// TwinCAT 3 PLC project Lectures
// ProgramVersion: 3.1.4024.0
// libraries:
//   Tc2_Standard, * (Beckhoff Automation GmbH)
//   Tc2_System, * (Beckhoff Automation GmbH)
//   Tc3_Module, * (Beckhoff Automation GmbH)
// project tree:
//   DUTs/ Motor.TcTLEO (not stored), Movement.TcTLEO, MovementDirection.TcTLEO (not stored), Recipe.TcDUT
//   GVLs/ Automatic.TcGVL, IO.TcGVL (not stored)
//   / PlcTask.TcTTO (not stored)
//   POUs/ AutomaticControl.TcPOU (not stored), CountCurrentPosition.TcPOU, ExecuteCurrentRecipe.TcPOU (not stored), Initialize.TcPOU, MakeNewRecipe.TcPOU (not stored), ManualControl.TcPOU, MAIN.TcPOU, MotorSelection.TcPOU (not stored), Recipe1.TcPOU (not stored), Recipe2.TcPOU, RestorePreviousAutomaticState.TcPOU, Safety.TcPOU (not stored)
//   POUs/Lectures%27 programs/ p00_true_false.TcPOU (not stored), p01_sequential.TcPOU (not stored), p02_clock.TcPOU (not stored), p03_SR1.TcPOU (not stored), p04_latch.TcPOU (not stored), p05_posEdge.TcPOU (not stored), p06_frontDetection.TcPOU (not stored), p07_memoryCell.TcPOU (not stored), p08_counter.TcPOU (not stored), p09_timers.TcPOU (not stored), p10_directionalInterlock.TcPOU (not stored), p11_logicalFunction.TcPOU (not stored), p12_controlLight.TcPOU (not stored)
//   POUs/RecipeFunctions/ Extension.TcPOU (not stored), Grip.TcPOU, Lifting.TcPOU, Rotation.TcPOU (not stored)
//   POUs/RestoreFunctions/ Restore.TcPOU
// real-time tasks:
//   TASK PlcTask1: cycle T#10ms, priority 21, ADS port 351
//   TASK PlcTask: cycle T#10ms, priority 20, ADS port 350
// I/O:
//   DEVICE Device 1 (EtherCAT), AmsNetId 172.31.192.1.2.1
//     Term 1 (EK1200) [EK1200-7000 EtherCAT Power supply (1,5A E-Bus)]
//       Term 2 (EL1859) [EL1859 8Ch. Dig. Input 24V, 3ms, 8Ch. Dig. Output 24V, 0.5A]
//       Term 3 (EL1859) [EL1859 8Ch. Dig. Input 24V, 3ms, 8Ch. Dig. Output 24V, 0.5A]
//       Term 4 (EL9011) [EL9011 End Terminal]
//   DEVICE Device 2 (NOV-DP-RAM) (disabled)
//   DEVICE Device 3 (CX7000), AmsNetId 172.31.192.1.4.1
//     Term 1 (CX7028) [CX7028-0000-0121]
//       modules: Module 1 (DIO_2x), Module 2 (Empty Module), Module 3 (DIO_2x), Module 4 (Empty Module), Module 5 (DI_2x), Module 6 (Empty Module), Module 7 (DI_2x), Module 8 (Empty Module)
// variable links:
//   Lectures/Lectures Instance <-> Device 1 (EtherCAT)/Term 1 (EK1200)/Term 2 (EL1859)
//     PlcTask Inputs/IO.EndExtensionSensor <-> Channel 3/Input
//     PlcTask Inputs/IO.EndGripSensor <-> Channel 7/Input
//     PlcTask Inputs/IO.EndLiftingSensor <-> Channel 5/Input
//     PlcTask Inputs/IO.EndRotationSensor <-> Channel 1/Input
//     PlcTask Inputs/IO.StepExtensionSwitch <-> Channel 4/Input
//     PlcTask Inputs/IO.StepGripSwitch <-> Channel 8/Input
//     PlcTask Inputs/IO.StepLiftingSwitch <-> Channel 6/Input
//     PlcTask Inputs/IO.StepRotatonSwitch <-> Channel 2/Input
//     PlcTask Outputs/IO.MotorExtension <-> Channel 12/Output
//     PlcTask Outputs/IO.MotorExtensionDirection <-> Channel 11/Output
//     PlcTask Outputs/IO.MotorGrip <-> Channel 16/Output
//     PlcTask Outputs/IO.MotorGripDirection <-> Channel 15/Output
//     PlcTask Outputs/IO.MotorLifting <-> Channel 14/Output
//     PlcTask Outputs/IO.MotorLiftingDirection <-> Channel 13/Output
//     PlcTask Outputs/IO.MotorRotation <-> Channel 10/Output
//     PlcTask Outputs/IO.MotorRotationDirection <-> Channel 9/Output
//   Lectures/Lectures Instance <-> Device 3 (CX7000)/Term 1 (CX7028)
//     PlcTask Inputs/IO.ButtonGreen <-> Module 3 (DIO_2x)/DIO_2x Input Channel 2/Input
//     PlcTask Inputs/IO.ButtonLowerLeft <-> Module 5 (DI_2x)/DI_2x Input Channel 1/Input
//     PlcTask Inputs/IO.ButtonLowerRight <-> Module 5 (DI_2x)/DI_2x Input Channel 2/Input
//     PlcTask Inputs/IO.ButtonRed <-> Module 1 (DIO_2x)/DIO_2x Input Channel 1/Input
//     PlcTask Inputs/IO.ButtonUpperLeft <-> Module 1 (DIO_2x)/DIO_2x Input Channel 2/Input
//     PlcTask Inputs/IO.ButtonUpperRight <-> Module 3 (DIO_2x)/DIO_2x Input Channel 1/Input
//     PlcTask Inputs/IO.Switch <-> Module 7 (DI_2x)/DI_2x Input Channel 1/Input
//     PlcTask Outputs/IO.LEDBlueLower <-> Module 3 (DIO_2x)/DIO_2x Output Channel 2/Output
//     PlcTask Outputs/IO.LEDBlueUpper <-> Module 1 (DIO_2x)/DIO_2x Output Channel 2/Output
//     PlcTask Outputs/IO.LEDGreen <-> Module 3 (DIO_2x)/DIO_2x Output Channel 1/Output
//     PlcTask Outputs/IO.LEDRed <-> Module 1 (DIO_2x)/DIO_2x Output Channel 1/Output

// ---- DUTs/Movement.TcTLEO
{attribute 'qualified_only'}
{attribute 'strict'}
TYPE Movement :
(
	ON := 1,
	OFF := 0
);
END_TYPE

// ---- DUTs/Recipe.TcDUT
TYPE Recipe :
STRUCT
	NoOfMovements: INT;
	MovementList: ARRAY[1..100] OF INT;
	MovementMotors: ARRAY[1..100] OF Motor;
END_STRUCT
END_TYPE

// ---- GVLs/Automatic.TcGVL
{attribute 'qualified_only'}
VAR_GLOBAL
	RCurrentlyMoving: BOOL;
	RotationPositionAuto: INT;
	RotationPositionCurrent: INT;
	SafetyRON: BOOL;
	
	LCurrentlyMoving: BOOL;
	LiftingPositionAuto: INT;
	LiftingPositionCurrent: INT;
	SafetyLON: BOOL;
	
	ECurrentlyMoving: BOOL;
	ExtensionPositionAuto: INT;
	ExtensionPositionCurrent: INT;
	SafetyEON: BOOL;
	
	GCurrentlyMoving: BOOL;
	GripPositionAuto: INT;
	GripPositionCurrent: INT;
	SafetyGON: BOOL;
	
	AllRestored: BOOL;
	
	Recipes: ARRAY[1..50] OF Recipe;
	RecipesIndex: INT := 3;
	CurrentRecipe: INT;
END_VAR

// ---- POUs/CountCurrentPosition.TcPOU
FUNCTION_BLOCK CountCurrentPosition
VAR_INPUT
END_VAR
VAR_OUTPUT
END_VAR
VAR
END_VAR

IF IO.Initialized THEN
	
	// COUNT ROTATION:
	IF IO.StepRotatonSwitch = 1 AND Automatic.RCurrentlyMoving THEN
		// away from the sensor:
		IF IO.MotorRotationDirection = 0 THEN
			IF (NOT IO.Switch) THEN		// in automatic mode
				IF IO.PreviousManualMode THEN	
					Automatic.RotationPositionCurrent := Automatic.RotationPositionCurrent + 1;
				ELSE	// to restore the state
					Automatic.RotationPositionCurrent := Automatic.RotationPositionCurrent + 1;
					Automatic.RotationPositionAuto := Automatic.RotationPositionAuto + 1;
				END_IF
			ELSE		// in manual mode
				Automatic.RotationPositionCurrent := Automatic.RotationPositionCurrent + 1;
			END_IF
		// towards the sensor:
		ELSE
			IF (NOT IO.Switch) THEN		// in automatic mode
				IF IO.PreviousManualMode THEN	
					Automatic.RotationPositionCurrent := Automatic.RotationPositionCurrent - 1;
				ELSE	// to restore the state
					Automatic.RotationPositionCurrent := Automatic.RotationPositionCurrent - 1;
					Automatic.RotationPositionAuto := Automatic.RotationPositionAuto - 1;
				END_IF
			ELSE		// in manual mode
				Automatic.RotationPositionCurrent := Automatic.RotationPositionCurrent - 1;
			END_IF
		END_IF
	END_IF
	
	// COUNT Extension:
	IF IO.StepExtensionSwitch = 1 AND Automatic.ECurrentlyMoving THEN
		// away from the sensor:
		IF IO.MotorExtensionDirection = 0 THEN
			IF (NOT IO.Switch) THEN		// in automatic mode
				IF IO.PreviousManualMode THEN
					Automatic.ExtensionPositionCurrent := Automatic.ExtensionPositionCurrent + 1;
				ELSE	// to restore the state
					Automatic.ExtensionPositionCurrent := Automatic.ExtensionPositionCurrent + 1;
					Automatic.ExtensionPositionAuto := Automatic.ExtensionPositionAuto + 1;
				END_IF
			ELSE		// in manual mode
				Automatic.ExtensionPositionCurrent := Automatic.ExtensionPositionCurrent + 1;
			END_IF
		// towards the sensor:
		ELSE
			IF (NOT IO.Switch) THEN		// in automatic mode
				IF IO.PreviousManualMode THEN	
					Automatic.ExtensionPositionCurrent := Automatic.ExtensionPositionCurrent - 1;
				ELSE	// to restore the state
					Automatic.ExtensionPositionCurrent := Automatic.ExtensionPositionCurrent - 1;
					Automatic.ExtensionPositionAuto := Automatic.ExtensionPositionAuto - 1;
				END_IF
			ELSE		// in manual mode
				Automatic.ExtensionPositionCurrent := Automatic.ExtensionPositionCurrent - 1;
			END_IF
		END_IF
	END_IF
	
	// COUNT Lifting:
	IF IO.StepLiftingSwitch = 1 AND Automatic.LCurrentlyMoving THEN
		// away from the sensor:
		IF IO.MotorLiftingDirection = 0 THEN
			IF (NOT IO.Switch) THEN		// in automatic mode
				IF IO.PreviousManualMode THEN
					Automatic.LiftingPositionCurrent := Automatic.LiftingPositionCurrent + 1;
				ELSE	// to restore the state
					Automatic.LiftingPositionCurrent := Automatic.LiftingPositionCurrent + 1;
					Automatic.LiftingPositionAuto := Automatic.LiftingPositionAuto + 1;
				END_IF
			ELSE		// in manual mode
				Automatic.LiftingPositionCurrent := Automatic.LiftingPositionCurrent + 1;
			END_IF
		// towards the sensor:
		ELSE
			IF (NOT IO.Switch) THEN		// in automatic mode
				IF IO.PreviousManualMode THEN
					Automatic.LiftingPositionCurrent := Automatic.LiftingPositionCurrent - 1;
				ELSE	// to restore the state
					Automatic.LiftingPositionAuto := Automatic.LiftingPositionAuto - 1;
					Automatic.LiftingPositionCurrent := Automatic.LiftingPositionCurrent - 1;
				END_IF
			ELSE		// in manual mode
				Automatic.LiftingPositionCurrent := Automatic.LiftingPositionCurrent - 1;
			END_IF
		END_IF
	END_IF
	
	// COUNT Grip:
	IF IO.StepGripSwitch = 1 AND Automatic.GCurrentlyMoving THEN
		IF IO.MotorGripDirection = 0 THEN
			IF (NOT IO.Switch) THEN		// in automatic mode
				IF IO.PreviousManualMode THEN
					Automatic.GripPositionCurrent := Automatic.GripPositionCurrent + 1;
				ELSE
					Automatic.GripPositionAuto := Automatic.GripPositionAuto + 1;
					Automatic.GripPositionCurrent := Automatic.GripPositionCurrent + 1;
				END_IF
			ELSE		// in manual mode
				Automatic.GripPositionCurrent := Automatic.GripPositionCurrent + 1;
			END_IF
		ELSE
			IF (NOT IO.Switch) THEN		// in automatic mode
				IF IO.PreviousManualMode THEN
					Automatic.GripPositionCurrent := Automatic.GripPositionCurrent - 1;
				ELSE
					Automatic.GripPositionAuto := Automatic.GripPositionAuto - 1;
					Automatic.GripPositionCurrent := Automatic.GripPositionCurrent - 1;
				END_IF
			ELSE		// in manual mode
				Automatic.GripPositionCurrent := Automatic.GripPositionCurrent - 1;
			END_IF
		END_IF
	END_IF
	
END_IF

END_FUNCTION_BLOCK

// ---- POUs/Initialize.TcPOU
PROGRAM Initialize
VAR
END_VAR

// go to the initial position (0,0,0,0)
IF NOT IO.Initialized THEN
	IF IO.EndRotationSensor THEN
		IO.MotorRotation := 0;
		IO.MotorRotationDirection := 0;
		Automatic.RCurrentlyMoving := FALSE;
	ELSE 
		IO.MotorRotationDirection := 1;
		Automatic.RCurrentlyMoving := TRUE;
		IO.MotorRotation := 1;
	END_IF
	
	IF IO.EndLiftingSensor THEN
		IO.MotorLifting := 0;
		IO.MotorLiftingDirection := 0;
		Automatic.LCurrentlyMoving := FALSE;
	ELSE 
		IO.MotorLiftingDirection := 1;
		Automatic.LCurrentlyMoving := TRUE;
		IO.MotorLifting := 1;
	END_IF
	
	IF IO.EndExtensionSensor THEN
		IO.MotorExtension := 0;
		IO.MotorExtensionDirection := 0;
		Automatic.ECurrentlyMoving := FALSE;
	ELSE 
		IO.MotorExtensionDirection := 1;
		Automatic.ECurrentlyMoving := TRUE;
		IO.MotorExtension := 1;
	END_IF
	
	IF IO.EndGripSensor THEN
		IO.MotorGrip := 0;
		IO.MotorGripDirection := 0;
		Automatic.GCurrentlyMoving := FALSE;
	ELSE 
		IO.MotorGripDirection := 1;
		Automatic.GCurrentlyMoving := TRUE;
		IO.MotorGrip := 1;
	END_IF
		
	IF IO.EndRotationSensor AND IO.EndLiftingSensor AND IO.EndExtensionSensor AND IO.EndGripSensor THEN
		Automatic.RCurrentlyMoving := FALSE;
		Automatic.ECurrentlyMoving := FALSE;
		Automatic.LCurrentlyMoving := FALSE;
		Automatic.GCurrentlyMoving := FALSE;
		IO.Initialized := TRUE;
		IO.PreviousManualMode := TRUE;
	END_IF
END_IF

END_PROGRAM

// ---- POUs/ManualControl.TcPOU
FUNCTION_BLOCK PUBLIC ManualControl
VAR_INPUT
	Switch: BOOL;
END_VAR
VAR
	ManualControl: BOOL;
	TimeForInterlockDelay: TIME := T#0.05S;
	ManualMode: BOOL;
	MotorSelection_1: MotorSelection;
	SelectedMotor: WORD;
	temp: TIME;
	LowerLeftInterlock: TOF;
	LowerLeft: BOOL;
	LowerRightInterlock: TOF;
	LowerRight: BOOL;
END_VAR
VAR_OUTPUT
	Output: BOOL;
END_VAR
VAR // added by the converter: edge detectors and wires of the graphical bodies
    _w1, _w2, _w3, _w4, _w5, _w6, _w7, _w8, _w9, _w10, _w11 : BOOL;
    _rt1, _rt2, _rt3 : R_TRIG;
    _ft1, _ft2, _ft3 : F_TRIG;
END_VAR

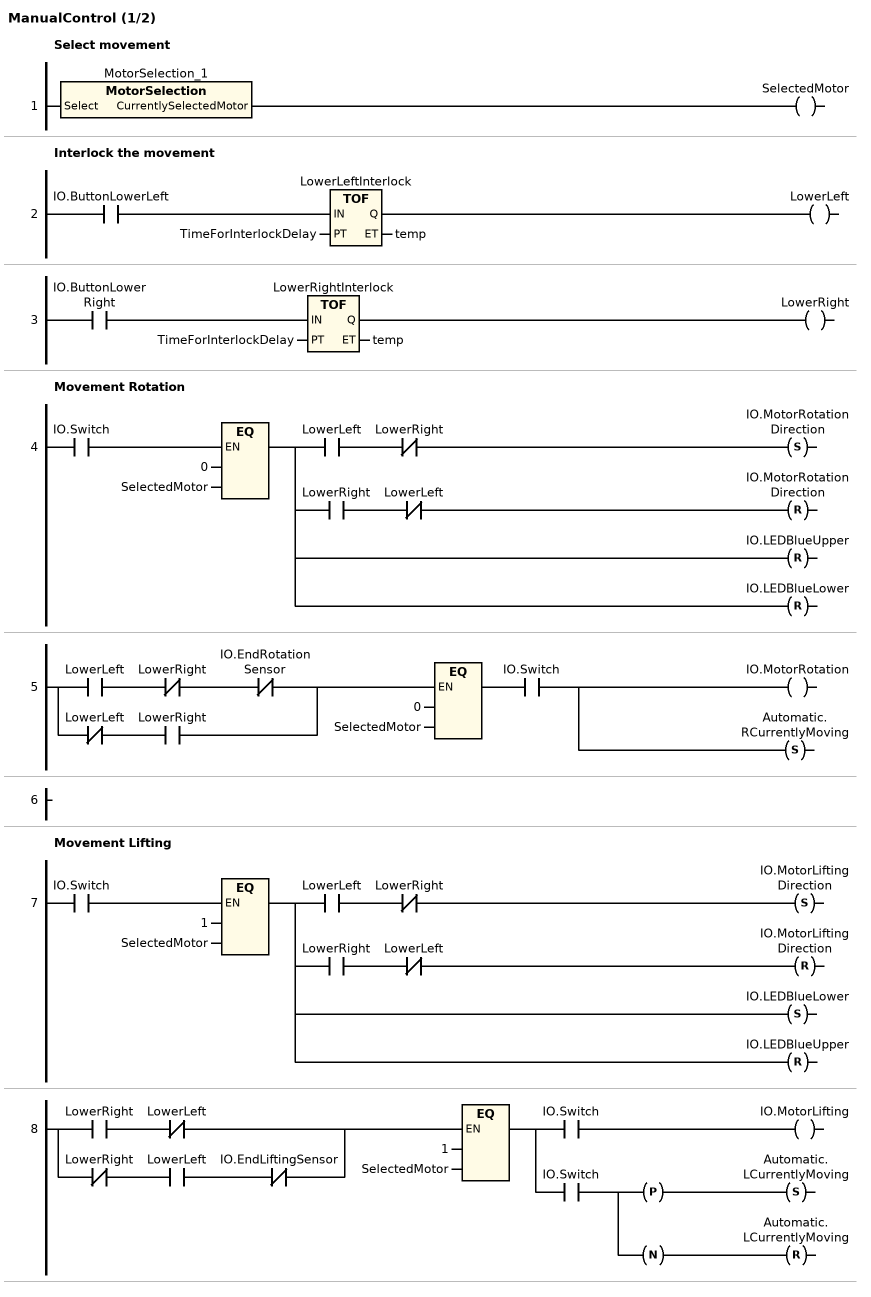
// NETWORK 1: Select movement
MotorSelection_1(Select := TRUE); // MotorSelection
SelectedMotor := MotorSelection_1.CurrentlySelectedMotor;

// NETWORK 2: Interlock the movement
LowerLeftInterlock(IN := IO.ButtonLowerLeft, PT := TimeForInterlockDelay, ET => temp); // TOF
LowerLeft := LowerLeftInterlock.Q;

// NETWORK 3
LowerRightInterlock(IN := IO.ButtonLowerRight, PT := TimeForInterlockDelay, ET => temp); // TOF
LowerRight := LowerRightInterlock.Q;

// NETWORK 4: Movement Rotation
_w1 := IO.Switch AND 0 = SelectedMotor;
IO.MotorRotationDirection S= _w1 AND LowerLeft AND NOT LowerRight;
IO.MotorRotationDirection R= _w1 AND LowerRight AND NOT LowerLeft;
IO.LEDBlueUpper R= _w1;
IO.LEDBlueLower R= _w1;

// NETWORK 5
_w2 := ((LowerLeft AND NOT LowerRight AND NOT IO.EndRotationSensor OR NOT LowerLeft AND LowerRight) AND 0 = SelectedMotor) AND IO.Switch;
IO.MotorRotation := _w2;
Automatic.RCurrentlyMoving S= _w2;

// NETWORK 6

// NETWORK 7: Movement Lifting
_w3 := IO.Switch AND 1 = SelectedMotor;
IO.MotorLiftingDirection S= _w3 AND LowerLeft AND NOT LowerRight;
IO.MotorLiftingDirection R= _w3 AND LowerRight AND NOT LowerLeft;
IO.LEDBlueLower S= _w3;
IO.LEDBlueUpper R= _w3;

// NETWORK 8
_w4 := (LowerRight AND NOT LowerLeft OR NOT LowerRight AND LowerLeft AND NOT IO.EndLiftingSensor) AND 1 = SelectedMotor;
IO.MotorLifting := _w4 AND IO.Switch;
_w5 := _w4 AND IO.Switch;
_rt1(CLK := _w5);
Automatic.LCurrentlyMoving S= _rt1.Q;
_ft1(CLK := _w5);
Automatic.LCurrentlyMoving R= _ft1.Q;

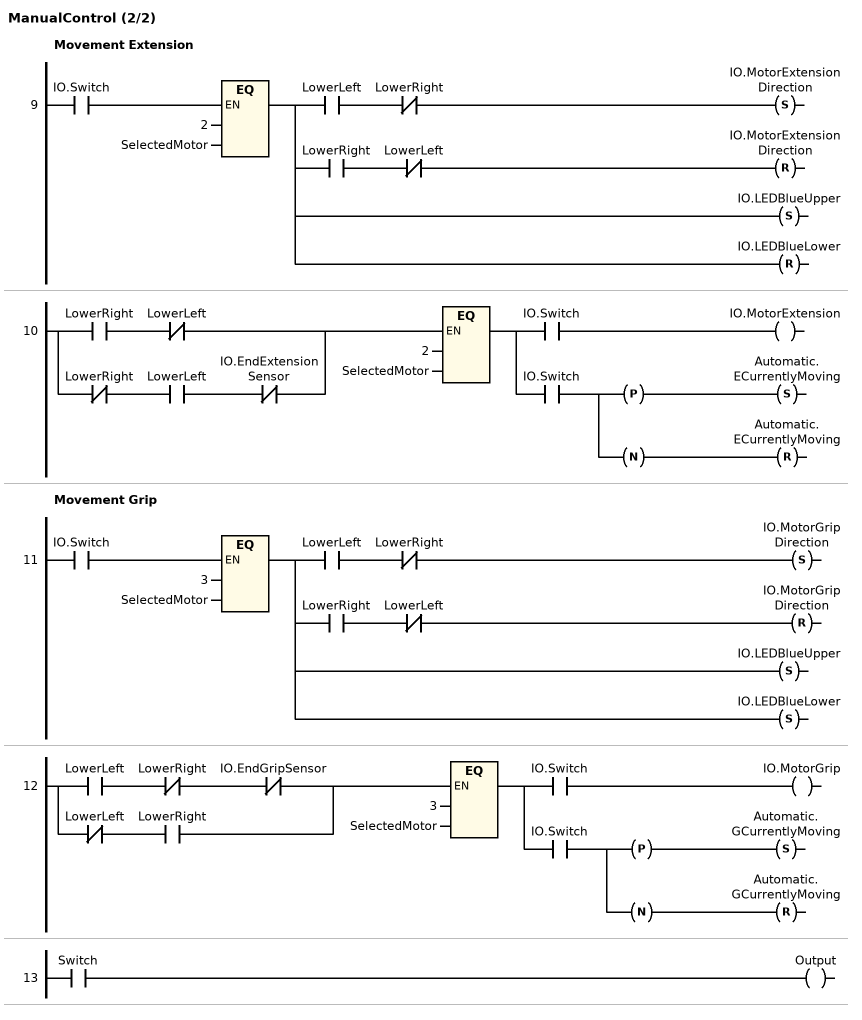
// NETWORK 9: Movement Extension
_w6 := IO.Switch AND 2 = SelectedMotor;
IO.MotorExtensionDirection S= _w6 AND LowerLeft AND NOT LowerRight;
IO.MotorExtensionDirection R= _w6 AND LowerRight AND NOT LowerLeft;
IO.LEDBlueUpper S= _w6;
IO.LEDBlueLower R= _w6;

// NETWORK 10
_w7 := (LowerRight AND NOT LowerLeft OR NOT LowerRight AND LowerLeft AND NOT IO.EndExtensionSensor) AND 2 = SelectedMotor;
IO.MotorExtension := _w7 AND IO.Switch;
_w8 := _w7 AND IO.Switch;
_rt2(CLK := _w8);
Automatic.ECurrentlyMoving S= _rt2.Q;
_ft2(CLK := _w8);
Automatic.ECurrentlyMoving R= _ft2.Q;

// NETWORK 11: Movement Grip
_w9 := IO.Switch AND 3 = SelectedMotor;
IO.MotorGripDirection S= _w9 AND LowerLeft AND NOT LowerRight;
IO.MotorGripDirection R= _w9 AND LowerRight AND NOT LowerLeft;
IO.LEDBlueUpper S= _w9;
IO.LEDBlueLower S= _w9;

// NETWORK 12
_w10 := (LowerLeft AND NOT LowerRight AND NOT IO.EndGripSensor OR NOT LowerLeft AND LowerRight) AND 3 = SelectedMotor;
IO.MotorGrip := _w10 AND IO.Switch;
_w11 := _w10 AND IO.Switch;
_rt3(CLK := _w11);
Automatic.GCurrentlyMoving S= _rt3.Q;
_ft3(CLK := _w11);
Automatic.GCurrentlyMoving R= _ft3.Q;

// NETWORK 13
Output := Switch;

END_FUNCTION_BLOCK

// ---- POUs/MAIN.TcPOU
PROGRAM MAIN
VAR
	ManualControl_0: ManualControl;
	AutomaticControl_0: AutomaticControl;
END_VAR

// Initially it goes to position (0,0,0,0) and initializes motors by Initialize PRG.
// There is Safety FB that keeps checking if motors are out of bounds.
// Motors are instantiated as global vars to retain their properties.
// CountCurrentPosition FB is the only place where we count position using the sensors.
// RestorePreviousAutomaticState is a FB that gets exectuted cyclically until all the motors are set to previous positions.
// AutomaticControl FB remembers which recipe is being executed and recipe remembers its state.
VAR // added by the converter: edge detectors and wires of the graphical bodies
    _ft1 : F_TRIG;
    _rt1 : R_TRIG;
    _w1 : BOOL;
END_VAR

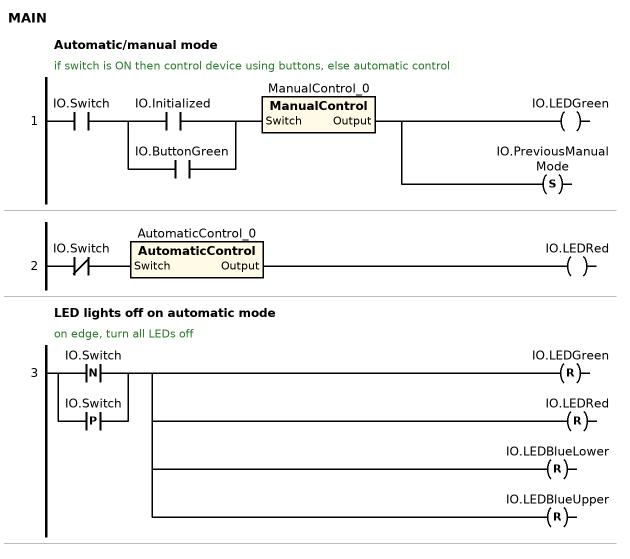
// NETWORK 1: Automatic/manual mode
// if switch is ON then control device using buttons, else automatic control
ManualControl_0(Switch := IO.Switch AND IO.Initialized OR IO.Switch AND IO.ButtonGreen); // ManualControl
IO.LEDGreen := ManualControl_0.Output;
IO.PreviousManualMode S= ManualControl_0.Output;

// NETWORK 2
AutomaticControl_0(Switch := NOT IO.Switch); // AutomaticControl
IO.LEDRed := AutomaticControl_0.Output;

// NETWORK 3: LED lights off on automatic mode
// on edge, turn all LEDs off
_ft1(CLK := IO.Switch);
_rt1(CLK := IO.Switch);
_w1 := _ft1.Q OR _rt1.Q;
IO.LEDGreen R= _w1;
IO.LEDRed R= _w1;
IO.LEDBlueLower R= _w1;
IO.LEDBlueUpper R= _w1;

END_PROGRAM

// ---- POUs/Recipe2.TcPOU
FUNCTION_BLOCK PUBLIC Recipe2
VAR_INPUT
	ExecutingRecipe2: BOOL;
	SuccesfullyEnded2: BOOL := FALSE;
END_VAR
VAR_OUTPUT
	SuccesfullyEnded: BOOL := FALSE;
END_VAR
VAR
	State: INT := 0;
	
	MinRotationPosition: INT := 0;
	InitialRotationPosition: INT := 140;
	
	MinLiftingPosition: INT := 0;
	InitialLiftingPosition: INT := 200;
	WoodInitialLiftingPosition: INT := 90;
	
	MinGripPosition: INT := 0;
	MaxGripPosition: INT := 160;

	MotorDirectionEnum: MovementDirection;	// for better clarity on the direction 0 and 1
	MovementEnum: Movement;	// for better clarity on the ON/OFF movement of the motors
END_VAR

IF ExecutingRecipe2 AND (NOT SuccesfullyEnded2) THEN	// we start executing recipe2 (again)
	SuccesfullyEnded := FALSE;
END_IF

IF NOT IO.Switch AND (NOT SuccesfullyEnded2) THEN
	
	IF State = 0 THEN
		State := Rotation(InitialRotationPosition, State);
		
	ELSIF State = 1 THEN
		State := Lifting(InitialLiftingPosition, State);
		
	ELSIF State = 2 THEN
		State := Grip(MaxGripPosition, State);
		
	ELSIF State = 3 THEN
		State := Lifting(MinLiftingPosition, State);
		
	ELSIF State = 4 THEN
		State := Rotation(MinRotationPosition, State);
		
	ELSIF State = 5 THEN
		State := Lifting(WoodInitialLiftingPosition, State);

	ELSIF State = 6 THEN
		State := Grip(MinGripPosition, State);
	
	ELSIF State = 7 THEN
		IO.Initialized := FALSE;
		SuccesfullyEnded := TRUE;
		State := 0;
		RETURN;
	END_IF
END_IF

END_FUNCTION_BLOCK

// ---- POUs/RecipeFunctions/Lifting.TcPOU
FUNCTION Lifting : INT
VAR_INPUT
	EndPosition: INT;
	State: INT;
END_VAR
VAR
	MovementEnum: Movement;
	NextState: INT;
	MotorDirectionEnum: MovementDirection;
END_VAR

IF Automatic.LiftingPositionAuto > EndPosition THEN
	MotorDirectionEnum := MovementDirection.TowardsSensor;
ELSE
	MotorDirectionEnum := MovementDirection.AwayFromSensor;
END_IF

IF MotorDirectionEnum = MovementDirection.TowardsSensor THEN
	IF Automatic.LiftingPositionAuto > EndPosition THEN
		IO.MotorLiftingDirection := (MotorDirectionEnum = MovementDirection.TowardsSensor);
		IF NOT Automatic.SafetyLON THEN
			Automatic.GCurrentlyMoving := TRUE;
			IO.MotorLifting := (MovementEnum = Movement.ON);
		END_IF
		NextState := State;
	ELSE
		IO.MotorLifting := (MovementEnum = Movement.OFF);
		NextState := State + 1;
		Automatic.LCurrentlyMoving := FALSE;
	END_IF
ELSE
	IF Automatic.LiftingPositionAuto < EndPosition THEN
		IO.MotorLiftingDirection := (MotorDirectionEnum = MovementDirection.AwayFromSensor);
		IF (NOT Automatic.SafetyLON) THEN
			Automatic.LCurrentlyMoving := TRUE;
			IO.MotorLifting := (MovementEnum = Movement.ON);
		END_IF
		NextState := State;
	ELSE
		IO.MotorLifting := (MovementEnum = Movement.OFF);
		NextState := State + 1;
		Automatic.LCurrentlyMoving := FALSE;
	END_IF
END_IF

Lifting := NextState;
RETURN;

END_FUNCTION

// ---- POUs/RecipeFunctions/Grip.TcPOU
FUNCTION Grip : INT
VAR_INPUT
	EndPosition: INT;
	State: INT;
END_VAR
VAR
	MovementEnum: Movement;
	NextState: INT;
	MotorDirectionEnum: MovementDirection;
END_VAR

IF Automatic.GripPositionAuto > EndPosition THEN
	MotorDirectionEnum := MovementDirection.TowardsSensor;
ELSE
	MotorDirectionEnum := MovementDirection.AwayFromSensor;
END_IF

IF MotorDirectionEnum = MovementDirection.TowardsSensor THEN
	IF Automatic.GripPositionAuto > EndPosition THEN
		IO.MotorGripDirection := (MotorDirectionEnum = MovementDirection.TowardsSensor);
		IF NOT Automatic.SafetyGON THEN
			Automatic.GCurrentlyMoving := TRUE;
			IO.MotorGrip := (MovementEnum = Movement.ON);
		END_IF
		NextState := State;
	ELSE
		IO.MotorGrip := (MovementEnum = Movement.OFF);
		NextState := State + 1;
		Automatic.GCurrentlyMoving := FALSE;
	END_IF
ELSE
	IF Automatic.GripPositionAuto < EndPosition THEN
		IO.MotorGripDirection := (MotorDirectionEnum = MovementDirection.AwayFromSensor);
		IF NOT Automatic.SafetyGON THEN
			Automatic.GCurrentlyMoving := TRUE;
			IO.MotorGrip := (MovementEnum = Movement.ON);
		END_IF
		NextState := State;
	ELSE
		IO.MotorGrip := (MovementEnum = Movement.OFF);
		NextState := State + 1;
		Automatic.GCurrentlyMoving := FALSE;
	END_IF
END_IF

Grip := NextState;
RETURN;

END_FUNCTION

// ---- POUs/RestoreFunctions/Restore.TcPOU
FUNCTION Restore : BOOL
VAR_INPUT
END_VAR
VAR
	MotorDirectionEnum: MovementDirection;	// for better clarity on the direction 0 and 1
	MovementEnum: Movement; // for better clarity on the ON/OFF movement of the motors
END_VAR
VAR_IN_OUT	// REFERENCES!
	Restored: BOOL;
	AUTOMATICPositionAuto: INT;
	AUTOMATICPositionCurrent: INT;
	AUTOMATICSafetyON: BOOL;
	AUTOMATICCurrentlyMoving: BOOL;
	IODirection: BOOL;	
	IOMotor: BOOL;
END_VAR

IF AUTOMATICPositionAuto - AUTOMATICPositionCurrent > 5 AND (NOT Restored) AND (NOT AUTOMATICSafetyON) THEN
	IODirection := (MotorDirectionEnum = MovementDirection.AwayFromSensor);
	AUTOMATICCurrentlyMoving := TRUE;
	IOMotor := (MovementEnum = Movement.ON);
	Restored := FALSE;
ELSIF AUTOMATICPositionCurrent - AUTOMATICPositionAuto > 5 AND (NOT Restored) AND (NOT AUTOMATICSafetyON) THEN
	IODirection := (MotorDirectionEnum = MovementDirection.TowardsSensor);
	AUTOMATICCurrentlyMoving := TRUE;
	IOMotor := (MovementEnum = Movement.ON);
	Restored := FALSE;
ELSE
	AUTOMATICCurrentlyMoving := FALSE;
	IOMotor := (MovementEnum = Movement.OFF);
	Restored := TRUE;
END_IF

Restore := Restored;
RETURN;	// Restored

END_FUNCTION

// ---- POUs/RestorePreviousAutomaticState.TcPOU
FUNCTION_BLOCK PUBLIC RestorePreviousAutomaticState
VAR_INPUT
END_VAR
VAR_OUTPUT
END_VAR
VAR
	RotationRestored: BOOL := FALSE;
	LiftingRestored: BOOL := FALSE;
	ExtensionRestored: BOOL := FALSE;
	GripRestored: BOOL := FALSE;
	DelayTimer: TON; // Timer instance
	
	MotorDirectionEnum: MovementDirection;	// for better clarity on the direction 0 and 1
	MovementEnum: Movement;	// for better clarity on the ON/OFF movement of the motors
END_VAR

IF IO.PreviousManualMode THEN
	Automatic.AllRestored := FALSE;
END_IF

// reset:
Restore(RotationRestored, Automatic.RotationPositionAuto, Automatic.RotationPositionCurrent, 
		Automatic.SafetyRON, Automatic.RCurrentlyMoving, IO.MotorRotationDirection, IO.MotorRotation);

Restore(LiftingRestored, Automatic.LiftingPositionAuto, Automatic.LiftingPositionCurrent, 
		Automatic.SafetyLON, Automatic.LCurrentlyMoving, IO.MotorLiftingDirection, IO.MotorLifting);

Restore(ExtensionRestored, Automatic.ExtensionPositionAuto, Automatic.ExtensionPositionCurrent,
		Automatic.SafetyEON, Automatic.ECurrentlyMoving, IO.MotorExtensionDirection, IO.MotorExtension);

Restore(GripRestored, Automatic.GripPositionAuto, Automatic.GripPositionCurrent,
		Automatic.SafetyGON, Automatic.GCurrentlyMoving, IO.MotorGripDirection, IO.MotorGrip);


// if all restored then go on to execute recipes in AutomaticControl:
IF RotationRestored AND LiftingRestored AND ExtensionRestored AND GripRestored THEN
	DelayTimer(IN := TRUE, PT := T#1S); // Start the timer with a n-second delay
	IF DelayTimer.Q THEN
		IO.PreviousManualMode := FALSE;
		Automatic.AllRestored := TRUE;
		
		RotationRestored := FALSE;
		ExtensionRestored := FALSE;
		LiftingRestored := FALSE;
		GripRestored := FALSE;
		Automatic.RCurrentlyMoving := FALSE;
		Automatic.ECurrentlyMoving := FALSE;
		Automatic.LCurrentlyMoving := FALSE;
		Automatic.GCurrentlyMoving := FALSE;
		DelayTimer(IN := FALSE); // Reset the timer
    END_IF
ELSE
    DelayTimer(IN := FALSE); // Ensure the timer is reset if the conditions are not met
END_IF

END_FUNCTION_BLOCK
